(* IEC 61131-3 sources: Industry-PLC-LLM/data/PLCBEAD_repo/PLCBEAD_PLCEmbed-main/PLC-BEAD/Source/GEB/building_DEW_RH, 1 file *)

(* ---- DEW_RH.ST ---- *)
FUNCTION SDD:REAL

	VAR_INPUT
		T :	REAL;
		ICE :	BOOL;
	END_VAR

	IF ice THEN
		SDD := 611.153 * EXP(22.4433 * T / (272.186 + T));
	ELSE
		SDD := 611.213 * EXP(17.5043 * T / (241.2 + T));
	END_IF;

END_FUNCTION

FUNCTION DEW_CON:REAL

	VAR_INPUT
		RH :	REAL;
		T :	REAL;
	END_VAR

	IF RH > 0.0 AND T > -50.0 THEN
		DEW_CON := 2.166824303E-2 * RH * SDD(T,FALSE)  / (T - -273.15);
	ELSE
		DEW_CON := 0.0;
	END_IF;

END_FUNCTION

FUNCTION DEW_RH:REAL

	VAR_INPUT
		VC :	REAL;
		T :	REAL;
	END_VAR

	DEW_RH := LIMIT(0.0, VC / DEW_CON(1.0, T), 100.0);

END_FUNCTION

PROGRAM program0
	VAR
		VC :	REAL;
		T :	REAL;
		CEIL5_OUT : REAL;
	END_VAR

  	CEIL5_OUT := DEW_RH(VC, T);
END_PROGRAM
